{attribute 'GeneratedUsingTerminal: EL2521-0000-1016'}
{attribute addProperty BoxType "EL2521-0000-1016"}
{attribute addProperty Id "PTO_StatusAT %I*PTO_Status_B6D696E07ENC_Status_compactAT %I*ENC_Status_compact_EA7A730E7PTO_ControlAT %Q*PTO_Control_392B4D2E5PTO_Target_compactAT %Q*PTO_Target_compact_5C359F7D2ENC_Control_compactAT %Q*ENC_Control_compact_245CB94B3WcStateAT %I*WcState_9091E0EB2InfoDataAT %I*InfoData_32EB74EA10"}
{attribute addProperty CRC "227618107"}
{attribute addProperty Size "36"}
TYPE EL2521_0D912D3B :
STRUCT
	{attribute addProperty Name "PTO_Status"}
	PTO_Status : PTO_Status_B6D696E0;
	{attribute addProperty Name "ENC_Status_compact"}
	ENC_Status_compact : ENC_Status_compact_EA7A730E;
	{attribute addProperty Name "PTO_Control"}
	PTO_Control : PTO_Control_392B4D2E;
	{attribute addProperty Name "PTO_Target_compact"}
	PTO_Target_compact : PTO_Target_compact_5C359F7D;
	{attribute addProperty Name "ENC_Control_compact"}
	ENC_Control_compact : ENC_Control_compact_245CB94B;
	{attribute addProperty Name "WcState"}
	WcState : WcState_9091E0EB;
	{attribute addProperty Name "InfoData"}
	InfoData : InfoData_32EB74EA;
END_STRUCT
END_TYPE

(* stored: Version 1.2.0.0, ProductVersion 3.1.4024.9
   DUT EL2521_0D912D3B: Id {02fffdbe-027f-4274-8863-295025e5f2e4} *)
